// TIA Portal V19 export
DATA_BLOCK "A0301_Fermi_P3"   // DB56
// stored: InstanceOfName A0301_Fermi_P3_FB, InstanceOfType FB
"A0301_Fermi_P3_FB"
   // VAR_INPUT
   //    AreaInterface : "AreaInterface";
   //    ZSI : "udt_ZoneSafetyInterface";
   //    DSI : "udt_DeviceSafetyInterface";
   //    DataIn : Struct
   //       OP_Rest_PB : Bool := FALSE;
   //       OP_Work_PB : Bool := FALSE;
   //    END_STRUCT;
   //    CIn : Struct
   //       Manager : "ValveMachine_Manager";
   //       SemiAut : Bool := FALSE;
   //       P2 : Struct
   //          Fermi : "ValveMachine_COut";
   //          Sollevatore : "ValveMachine_COut";
   //       END_STRUCT;
   //       Trasporto : "SpeedMachine_COut";
   //    END_STRUCT;
   //    Config : Struct
   //       Fermi : Array[1..6] of "ValveMachine_Config";
   //       DelayMissingCondition : Time := T#3S;
   //    END_STRUCT;
   // END_VAR
   // VAR_OUTPUT
   //    MachineInterface : "MachineInterface";
   //    COut : Struct
   //       Fermi : "ValveMachine_COut";
   //    END_STRUCT;
   // END_VAR
   // VAR
   //    Alarm : Struct
   //       Fermi : Array[1..6] of "ValveAlr";
   //    END_STRUCT;
   //    Warning : Struct
   //       OP_REST_MissingCnd : Bool := FALSE;
   //       OP_WORK_MissingCnd : Bool := FALSE;
   //       Fermi : Array[1..6] of "ValveMachine_Wng";
   //    END_STRUCT;
   //    HMI : Struct
   //       Selection : Array[1..6] of Bool;
   //       FermiSts { S7_SetPoint := 'True'} : "UDT_HMI-Sts_ValvePosA0301";
   //       B_ResetShiftDone : Bool := FALSE;
   //    END_STRUCT;
   //    Sts : Struct
   //       Fermi_AlarmPresence : Bool := FALSE;
   //       OP_CanMoveFreely : Bool := TRUE;
   //       OP_Rest_Cnd : Bool := FALSE;
   //       Op_Work_Cnd : Bool := FALSE;
   //    END_STRUCT;
   //    Ctrl : Struct
   //       OP_Rest_Man : Bool := FALSE;
   //       OP_Work_Man : Bool := FALSE;
   //       OP_Rest_Aut : Bool := FALSE;
   //       OP_Work_Aut : Bool := FALSE;
   //       OP_Rest : Bool := FALSE;
   //       OP_Work : Bool := FALSE;
   //    END_STRUCT;
   //    Fermi { S7_SetPoint := 'True'} : Array[1..6] of "ValveMachine_FB";
   //    AUX : Struct
   //       OP_Rest_PB : Bool := FALSE;
   //       OP_Work_PB : Bool := FALSE;
   //    END_STRUCT;
   //    TON_OP_REST_MissingCnd { S7_SetPoint := 'True'} : TON_TIME;
   //    TON_OP_WORK_MissingCnd { S7_SetPoint := 'True'} : TON_TIME;
   // END_VAR
BEGIN
   AreaInterface.EStop := FALSE;
   AreaInterface.Man := TRUE;
   AreaInterface.Aut := FALSE;
   AreaInterface.Cycle := FALSE;
   AreaInterface.StopInPhase := FALSE;
   AreaInterface.StopProgrammed := FALSE;
   AreaInterface.RstAlarms := FALSE;
   AreaInterface.ManOneShot := FALSE;
   AreaInterface.AutOneShot := FALSE;
   AreaInterface.CycleOneShot := FALSE;
   AreaInterface.CheckAutReady := FALSE;
   ZSI.Door_NormalStop := FALSE;
   ZSI.Door_SafeStop := FALSE;
   ZSI.Door_Opened := FALSE;
   ZSI.Door_EntryEnable := FALSE;
   DSI.SafeStop := FALSE;
   DSI.PowerEnable := TRUE;
   DSI.DevicesInSafeState := FALSE;
   CIn.Manager.EnableStopDoorOpeningReq := FALSE;
   CIn.Manager.EnableStopInPhase := FALSE;
   CIn.Manager.EnableStopProgrammed := FALSE;
   CIn.Manager.Control_ON := FALSE;
   CIn.Manager.Rest := FALSE;
   CIn.Manager.Work := FALSE;
   CIn.P2.Fermi.CtrlSafe := FALSE;
   CIn.P2.Fermi.Standstill := TRUE;
   CIn.P2.Fermi.ReqOilPressure := FALSE;
   CIn.P2.Fermi.Rest_CheckNext := FALSE;
   CIn.P2.Fermi.Work_CheckNext := FALSE;
   CIn.P2.Fermi.Rest := FALSE;
   CIn.P2.Fermi.Work := FALSE;
   CIn.P2.Sollevatore.CtrlSafe := FALSE;
   CIn.P2.Sollevatore.Standstill := TRUE;
   CIn.P2.Sollevatore.ReqOilPressure := FALSE;
   CIn.P2.Sollevatore.Rest_CheckNext := FALSE;
   CIn.P2.Sollevatore.Work_CheckNext := FALSE;
   CIn.P2.Sollevatore.Rest := FALSE;
   CIn.P2.Sollevatore.Work := FALSE;
   CIn.Trasporto.Infeed_ReqON := FALSE;
   CIn.Trasporto.CtrlSafe := FALSE;
   CIn.Trasporto.Standstill := TRUE;
   CIn.Trasporto.Bwd_CheckNext := FALSE;
   CIn.Trasporto.Fwd_CheckNext := FALSE;
   CIn.Trasporto.Bwd_VelZero := FALSE;
   CIn.Trasporto.Bwd_Running := FALSE;
   CIn.Trasporto.Fwd_VelZero := FALSE;
   CIn.Trasporto.Fwd_Running := FALSE;
   CIn.Trasporto.ActualVelocity := 0.0;
   CIn.Trasporto.TargetVelocity := 0.0;
   CIn.Trasporto.MaxVelocity := 39597.8;
   Config.Fermi[1..6].DelayPressureRunningTimeout := T#3S;
   Config.Fermi[1..6].DelayMissingCondition := T#3S;
   Config.Fermi[1..6].Rest_LsQty := 1;
   Config.Fermi[1..6].Work_LsQty := 0;
   Config.Fermi[1..6].Rest_RetainAut := FALSE;
   Config.Fermi[1..6].Work_RetainAut := FALSE;
   Config.Fermi[1..6].V.RestLimSwitchExist := TRUE;
   Config.Fermi[1..6].V.WorkLimSwitchExist := FALSE;
   Config.Fermi[1..6].V.CheckOilInPressure := FALSE;
   Config.Fermi[1..6].V.CutRestWhenIsAtRest := TRUE;
   Config.Fermi[1..6].V.CutWorkWhenIsAtWork := TRUE;
   Config.Fermi[1..6].V.RestTime := T#2S;
   Config.Fermi[1..6].V.WorkTime := T#2S;
   Config.Fermi[1..6].V.RestTimeOut := T#1H;
   Config.Fermi[1..6].V.WorkTimeOut := T#1H;
   MachineInterface.AutReady := FALSE;
   MachineInterface.Aborting := FALSE;
   MachineInterface.AckStopInPhase := FALSE;
   MachineInterface.AckStopProgrammed := FALSE;
   MachineInterface.MotionsStandStill := TRUE;
   MachineInterface.AlarmsPresence := FALSE;
   MachineInterface.WarningPresence := FALSE;
   COut.Fermi.CtrlSafe := FALSE;
   COut.Fermi.Standstill := TRUE;
   COut.Fermi.ReqOilPressure := FALSE;
   COut.Fermi.Rest_CheckNext := FALSE;
   COut.Fermi.Work_CheckNext := FALSE;
   COut.Fermi.Rest := FALSE;
   COut.Fermi.Work := FALSE;
   Alarm.Fermi[1..6].TimeOutRest := FALSE;
   Alarm.Fermi[1..6].TimeOutWork := FALSE;
   Alarm.Fermi[1..6].LimitSwitches := FALSE;
   Warning.Fermi[1..6].NotAutReady := FALSE;
   Warning.Fermi[1..6].PressureRunning_Timeout := FALSE;
   Warning.Fermi[1..6].Rest_MissingExtEnable := FALSE;
   Warning.Fermi[1..6].Work_MissingExtEnable := FALSE;
   Warning.Fermi[1].Missing_Rest_Ls_ON[1..8] := FALSE;
   Warning.Fermi[2].Missing_Rest_Ls_ON[1..8] := FALSE;
   Warning.Fermi[3].Missing_Rest_Ls_ON[1..8] := FALSE;
   Warning.Fermi[4].Missing_Rest_Ls_ON[1..8] := FALSE;
   Warning.Fermi[5].Missing_Rest_Ls_ON[1..8] := FALSE;
   Warning.Fermi[6].Missing_Rest_Ls_ON[1..8] := FALSE;
   Warning.Fermi[1].Missing_Work_Ls_ON[1..8] := FALSE;
   Warning.Fermi[2].Missing_Work_Ls_ON[1..8] := FALSE;
   Warning.Fermi[3].Missing_Work_Ls_ON[1..8] := FALSE;
   Warning.Fermi[4].Missing_Work_Ls_ON[1..8] := FALSE;
   Warning.Fermi[5].Missing_Work_Ls_ON[1..8] := FALSE;
   Warning.Fermi[6].Missing_Work_Ls_ON[1..8] := FALSE;
   HMI.Selection[1..6] := TRUE;
   HMI.FermiSts.Standstill := TRUE;
   HMI.FermiSts.Rest := FALSE;
   HMI.FermiSts.Work := FALSE;
   HMI.FermiSts.AlarmPresence := FALSE;
   Fermi[1..6].AreaInterface.EStop := FALSE;
   Fermi[1..6].AreaInterface.Man := TRUE;
   Fermi[1..6].AreaInterface.Aut := FALSE;
   Fermi[1..6].AreaInterface.Cycle := FALSE;
   Fermi[1..6].AreaInterface.StopInPhase := FALSE;
   Fermi[1..6].AreaInterface.StopProgrammed := FALSE;
   Fermi[1..6].AreaInterface.RstAlarms := FALSE;
   Fermi[1..6].AreaInterface.ManOneShot := FALSE;
   Fermi[1..6].AreaInterface.AutOneShot := FALSE;
   Fermi[1..6].AreaInterface.CycleOneShot := FALSE;
   Fermi[1..6].AreaInterface.CheckAutReady := FALSE;
   Fermi[1..6].ZSI.Door_NormalStop := FALSE;
   Fermi[1..6].ZSI.Door_SafeStop := FALSE;
   Fermi[1..6].ZSI.Door_Opened := FALSE;
   Fermi[1..6].ZSI.Door_EntryEnable := FALSE;
   Fermi[1..6].DSI.SafeStop := FALSE;
   Fermi[1..6].DSI.PowerEnable := TRUE;
   Fermi[1..6].DSI.DevicesInSafeState := FALSE;
   Fermi[1..6].DataIn.PB.Rest := FALSE;
   Fermi[1..6].DataIn.PB.Work := FALSE;
   Fermi[1..6].DataIn.PB.StartStop := FALSE;
   Fermi[1].DataIn.Rest_Ls[1] := TRUE;
   Fermi[1].DataIn.Rest_Ls[2..8] := FALSE;
   Fermi[2].DataIn.Rest_Ls[1] := TRUE;
   Fermi[2].DataIn.Rest_Ls[2..8] := FALSE;
   Fermi[3].DataIn.Rest_Ls[1] := TRUE;
   Fermi[3].DataIn.Rest_Ls[2..8] := FALSE;
   Fermi[4].DataIn.Rest_Ls[1] := TRUE;
   Fermi[4].DataIn.Rest_Ls[2..8] := FALSE;
   Fermi[5].DataIn.Rest_Ls[1] := TRUE;
   Fermi[5].DataIn.Rest_Ls[2..8] := FALSE;
   Fermi[6].DataIn.Rest_Ls[1] := TRUE;
   Fermi[6].DataIn.Rest_Ls[2..8] := FALSE;
   Fermi[1].DataIn.Work_Ls[1..8] := FALSE;
   Fermi[2].DataIn.Work_Ls[1..8] := FALSE;
   Fermi[3].DataIn.Work_Ls[1..8] := FALSE;
   Fermi[4].DataIn.Work_Ls[1..8] := FALSE;
   Fermi[5].DataIn.Work_Ls[1..8] := FALSE;
   Fermi[6].DataIn.Work_Ls[1..8] := FALSE;
   Fermi[1..6].Cin.Manager.EnableStopDoorOpeningReq := FALSE;
   Fermi[1..6].Cin.Manager.EnableStopInPhase := FALSE;
   Fermi[1..6].Cin.Manager.EnableStopProgrammed := FALSE;
   Fermi[1..6].Cin.Manager.Control_ON := FALSE;
   Fermi[1..6].Cin.Manager.Rest := FALSE;
   Fermi[1..6].Cin.Manager.Work := FALSE;
   Fermi[1..6].Cin.PressureRunning := FALSE;
   Fermi[1..6].Cin.Rest_ExtEnable := TRUE;
   Fermi[1..6].Cin.Work_ExtEnable := TRUE;
   Fermi[1..6].Cin.ExternalAlarms := FALSE;
   Fermi[1..6].Config.DelayPressureRunningTimeout := T#3S;
   Fermi[1..6].Config.DelayMissingCondition := T#3S;
   Fermi[1..6].Config.Rest_LsQty := 1;
   Fermi[1..6].Config.Work_LsQty := 0;
   Fermi[1..6].Config.Rest_RetainAut := FALSE;
   Fermi[1..6].Config.Work_RetainAut := FALSE;
   Fermi[1..6].Config.V.RestLimSwitchExist := TRUE;
   Fermi[1..6].Config.V.WorkLimSwitchExist := FALSE;
   Fermi[1..6].Config.V.CheckOilInPressure := FALSE;
   Fermi[1..6].Config.V.CutRestWhenIsAtRest := TRUE;
   Fermi[1..6].Config.V.CutWorkWhenIsAtWork := TRUE;
   Fermi[1..6].Config.V.RestTime := T#2S;
   Fermi[1..6].Config.V.WorkTime := T#2S;
   Fermi[1..6].Config.V.RestTimeOut := T#1H;
   Fermi[1..6].Config.V.WorkTimeOut := T#1H;
   Fermi[1..6].MachineInterface.AutReady := FALSE;
   Fermi[1..6].MachineInterface.Aborting := FALSE;
   Fermi[1..6].MachineInterface.AckStopInPhase := FALSE;
   Fermi[1..6].MachineInterface.AckStopProgrammed := FALSE;
   Fermi[1..6].MachineInterface.MotionsStandStill := TRUE;
   Fermi[1..6].MachineInterface.AlarmsPresence := FALSE;
   Fermi[1..6].MachineInterface.WarningPresence := FALSE;
   Fermi[1..6].COut.CtrlSafe := FALSE;
   Fermi[1..6].COut.Standstill := TRUE;
   Fermi[1..6].COut.ReqOilPressure := FALSE;
   Fermi[1..6].COut.Rest_CheckNext := FALSE;
   Fermi[1..6].COut.Work_CheckNext := FALSE;
   Fermi[1..6].COut.Rest := TRUE;
   Fermi[1..6].COut.Work := FALSE;
   Fermi[1..6].DataOut.RestSolenoid := FALSE;
   Fermi[1..6].DataOut.WorkSolenoid := FALSE;
   Fermi[1..6].Sts.Standstill := TRUE;
   Fermi[1..6].Sts.AlarmsPresence := FALSE;
   Fermi[1..6].Sts.WarningsPresence := FALSE;
   Fermi[1..6].Sts.Rest_Cnd := TRUE;
   Fermi[1..6].Sts.Work_Cnd := TRUE;
   Fermi[1..6].Ctrl.StopDueDoorOpeningRequest := FALSE;
   Fermi[1..6].Ctrl.StopInPhase := FALSE;
   Fermi[1..6].Ctrl.StopProgrammed := FALSE;
   Fermi[1..6].Ctrl.StopAborting := FALSE;
   Fermi[1..6].Ctrl.Work := FALSE;
   Fermi[1..6].Ctrl.Rest := FALSE;
   Fermi[1..6].Ctrl.Rest_Man := FALSE;
   Fermi[1..6].Ctrl.Work_Man := FALSE;
   Fermi[1..6].Ctrl.Rest_Aut := FALSE;
   Fermi[1..6].Ctrl.Work_Aut := FALSE;
   Fermi[1..6].V.ValveCtrl.SafeStop := FALSE;
   Fermi[1..6].V.ValveCtrl.Rst := FALSE;
   Fermi[1..6].V.ValveCtrl.MoveRest := FALSE;
   Fermi[1..6].V.ValveCtrl.MoveWork := FALSE;
   Fermi[1..6].V.RestLimitSwitch := TRUE;
   Fermi[1..6].V.WorkLimitSwitch := FALSE;
   Fermi[1..6].V.OilInPressure := FALSE;
   Fermi[1..6].V.Simulation := FALSE;
   Fermi[1..6].V.Config.RestLimSwitchExist := TRUE;
   Fermi[1..6].V.Config.WorkLimSwitchExist := FALSE;
   Fermi[1..6].V.Config.CheckOilInPressure := FALSE;
   Fermi[1..6].V.Config.CutRestWhenIsAtRest := TRUE;
   Fermi[1..6].V.Config.CutWorkWhenIsAtWork := TRUE;
   Fermi[1..6].V.Config.RestTime := T#2S;
   Fermi[1..6].V.Config.WorkTime := T#2S;
   Fermi[1..6].V.Config.RestTimeOut := T#1H;
   Fermi[1..6].V.Config.WorkTimeOut := T#1H;
   Fermi[1..6].V.ValveSts.AlarmPresence := FALSE;
   Fermi[1..6].V.ValveSts.RestPermit := TRUE;
   Fermi[1..6].V.ValveSts.RestInProgress := FALSE;
   Fermi[1..6].V.ValveSts.IsAtRest := TRUE;
   Fermi[1..6].V.ValveSts.WorkPermit := TRUE;
   Fermi[1..6].V.ValveSts.WorkInProgress := FALSE;
   Fermi[1..6].V.ValveSts.IsAtWork := FALSE;
   Fermi[1..6].V.ValveSts.StandStill := TRUE;
   Fermi[1..6].V.RestSolenoid := FALSE;
   Fermi[1..6].V.WorkSolenoid := FALSE;
   Fermi[1..6].V.ReqOilPressure := FALSE;
   Fermi[1..6].V.IsAtRest := TRUE;
   Fermi[1..6].V.IsAtWork := FALSE;
   Fermi[1..6].V.Ctrl.RestReq := FALSE;
   Fermi[1..6].V.Ctrl.WorkReq := FALSE;
   Fermi[1..6].V.Ctrl.RestSolenoid := FALSE;
   Fermi[1..6].V.Ctrl.WorkSolenoid := FALSE;
   Fermi[1..6].V.tonRest.PT := T#2S;
   Fermi[1..6].V.tonRest.IN := TRUE;
   Fermi[1..6].V.tonWork.PT := T#0MS;
   Fermi[1..6].V.tonWork.IN := FALSE;
   Fermi[1..6].V.tonTimeOutRest.PT := T#0MS;
   Fermi[1..6].V.tonTimeOutRest.IN := FALSE;
   Fermi[1..6].V.tonTimeOutWork.PT := T#0MS;
   Fermi[1..6].V.tonTimeOutWork.IN := FALSE;
   Fermi[1..6].TON_NoPendingCmd.PT := T#500MS;
   Fermi[1..6].TON_NoPendingCmd.IN := TRUE;
   Fermi[1..6].TON_Rest_MissingExtEnable.PT := T#0MS;
   Fermi[1..6].TON_Rest_MissingExtEnable.IN := FALSE;
   Fermi[1..6].TON_Work_MissingExtEnable.PT := T#0MS;
   Fermi[1..6].TON_Work_MissingExtEnable.IN := FALSE;
   Fermi[1..6].TON_PressureRunning_Timeout.PT := T#0MS;
   Fermi[1..6].TON_PressureRunning_Timeout.IN := FALSE;
   Fermi[1..6].Aux.Pb_Rest := FALSE;
   Fermi[1..6].Aux.Pb_Work := FALSE;
   Fermi[1..6].Aux.Pb_StartStop := FALSE;
   TON_OP_REST_MissingCnd.PT := T#0MS;
   TON_OP_REST_MissingCnd.IN := FALSE;
   TON_OP_WORK_MissingCnd.PT := T#0MS;
   TON_OP_WORK_MissingCnd.IN := FALSE;
END_DATA_BLOCK
